{attribute 'qualified_only'}
{attribute 'strict'}
{attribute 'to_string'}
TYPE E_HE_SATT_RoundingMode :
(
    FLOOR_WITHIN_TOLERANCE := 0,
    CEIL,
    FLOOR,
    CLOSEST,
    CEIL_WITHIN_TOLERANCE,
    CLOSEST_WITHIN_TOLERANCE
) UINT;
END_TYPE

(* stored: Version 1.1.0.1
   DUT E_HE_SATT_RoundingMode: Id {39f668eb-3f39-4c39-b199-6ea8f785627d} *)
